// TIA Portal project "2020-11-06_gestioneMotoreJogSS" (V16)
// Programma che gestisce la ventilazione di un motore

(* hardware
DEVICE "Stazione SIMATIC 1200_1"  S71200.Device
   slot 0: "Telaio di montaggio S7-1200"  Rack  V1.0
   slot 1: "PLC_1"  CPU 1215C DC/DC/DC  6ES7 215-1AG40-0XB0  V4.2
*)

// ===== PLC "PLC_1"  CPU 1215C DC/DC/DC =====

VAR_GLOBAL   // PLC tag table "Tabella delle variabili standard"
   "ventA_f" AT %I0.0 : Bool;
   "ventB_f" AT %I0.1 : Bool;
   "ventC_f" AT %I0.2 : Bool;
   "pulsanteJog_f" AT %I0.3 : Bool;
   "pulsanteStart_f" AT %I0.4 : Bool;
   "pulsanteStop_f" AT %I0.5 : Bool;
   "modoJog_f" AT %I0.6 : Bool;
   "motore" AT %Q0.0 : Bool;
   "ventilaz_NOOK" AT %Q0.1 : Bool;
   "modoSS_f" AT %I0.7 : Bool;
   "out2" AT %Q0.2 : Bool;
   "out3" AT %Q0.3 : Bool;
   "out4" AT %Q0.4 : Bool;
   "sempre vero" AT %M6.0 : Bool;   // bit sempre vero
   "uscite byte" AT %QB0 : Byte;   // Uscite fisiche
   "uscite memorie" AT %MB1 : Byte;   // uscite memorie da usare come ingressi
   "out4_M" AT %M1.4 : Bool;
   "out3_M" AT %M1.3 : Bool;
   "out2_M" AT %M1.2 : Bool;
   "ventilaz_NOOK_M" AT %M1.1 : Bool;
   "motore_M" AT %M1.0 : Bool;
   "ingressi byte" AT %IB0 : Byte;   // Ingressi fisici
   "ingressi memorie" AT %MB0 : Byte;   // Ingressi Na non filtrati
   "in0_na" AT %M0.0 : Bool;
   "in1_na" AT %M0.1 : Bool;
   "in2_na" AT %M0.2 : Bool;
   "in3_na" AT %M0.3 : Bool;
   "in4_na" AT %M0.4 : Bool;
   "in5_na" AT %M0.5 : Bool;
   "in6_na" AT %M0.6 : Bool;
   "in7_na" AT %M0.7 : Bool;
   "out5" AT %Q0.5 : Bool;
   "out6" AT %Q0.6 : Bool;
   "out7" AT %Q0.7 : Bool;
   "out5_M" AT %M1.5 : Bool;
   "out6_M" AT %M1.6 : Bool;
   "out7_M" AT %M1.7 : Bool;
   "ingressi memorie filtrato" AT %MB2 : Byte;
   "ventA" AT %M2.0 : Bool;
   "ventB" AT %M2.1 : Bool;
   "ventC" AT %M2.2 : Bool;
   "pulsanteJog" AT %M2.3 : Bool;
   "pulsanteStart" AT %M2.4 : Bool;
   "pulsanteStop" AT %M2.5 : Bool;
   "modoJog" AT %M2.6 : Bool;
   "modoSS" AT %M2.7 : Bool;
   "ingressi memorie_p" AT %MB3 : Byte;
   "in0_p" AT %M3.0 : Bool;
   "in1_p" AT %M3.1 : Bool;
   "in2_p" AT %M3.2 : Bool;
   "in3_p" AT %M3.3 : Bool;
   "pulsanteStart_p" AT %M3.4 : Bool;
   "pulsanteStop_p" AT %M3.5 : Bool;
   "in6_p" AT %M3.6 : Bool;
   "in7_p" AT %M3.7 : Bool;
   "ingressi_memorie_var_p" AT %MB4 : Byte;
   "in0_var_p" AT %M4.0 : Bool;
   "in1_var_p" AT %M4.1 : Bool;
   "in2_var_p" AT %M4.2 : Bool;
   "in3_var_p" AT %M4.3 : Bool;
   "in4_var_p" AT %M4.4 : Bool;
   "in5_var_p" AT %M4.5 : Bool;
   "in6_var_p" AT %M4.6 : Bool;
   "in7_var_p" AT %M4.7 : Bool;
   "ventilazione_OK" AT %M10.0 : Bool;
   "modoJog_OK" AT %M10.1 : Bool;
   "modoSS_OK" AT %M10.2 : Bool;
   "motoreJog" AT %M10.3 : Bool;
   "motoreSS" AT %M10.4 : Bool;
END_VAR

VAR_GLOBAL CONSTANT   // PLC tag table "Tabella delle variabili standard"
   "maschera NCNA" : Byte := B#2#00100100;   // mettere a 1 i bit NC
   "filtro in0" : Time := T#500ms;
   "filtro in1" : Time := T#500ms;
   "filtro in2" : Time := T#500ms;
   "filtro in3" : Time := T#200ms;
   "filtro in4" : Time := T#500ms;
   "filtro in5" : Time := T#100ms;
   "filtro in6" : Time := T#1s;
   "filtro in7" : Time := T#1s;
   "Maschera Out Reset" : Byte := B#2#00000000;
END_VAR

// folder: System blocks/Program resources

DATA_BLOCK "filtro_in0"   // DB1
{ S7_Optimized_Access := 'TRUE' }
AUTHOR : Simatic
FAMILY : IEC
NAME : IEC_TMR
VERSION : 1.0
// stored: InstanceOfName IEC_TIMER
"IEC_TIMER"
BEGIN
END_DATA_BLOCK

DATA_BLOCK "filtro_in1"   // DB2
{ S7_Optimized_Access := 'TRUE' }
AUTHOR : Simatic
FAMILY : IEC
NAME : IEC_TMR
VERSION : 1.0
// stored: InstanceOfName IEC_TIMER
"IEC_TIMER"
BEGIN
END_DATA_BLOCK

DATA_BLOCK "filtro_in2"   // DB3
{ S7_Optimized_Access := 'TRUE' }
AUTHOR : Simatic
FAMILY : IEC
NAME : IEC_TMR
VERSION : 1.0
// stored: InstanceOfName IEC_TIMER
"IEC_TIMER"
BEGIN
END_DATA_BLOCK

DATA_BLOCK "filtro_in3"   // DB4
{ S7_Optimized_Access := 'TRUE' }
AUTHOR : Simatic
FAMILY : IEC
NAME : IEC_TMR
VERSION : 1.0
// stored: InstanceOfName IEC_TIMER
"IEC_TIMER"
BEGIN
END_DATA_BLOCK

DATA_BLOCK "filtro_in4"   // DB5
{ S7_Optimized_Access := 'TRUE' }
AUTHOR : Simatic
FAMILY : IEC
NAME : IEC_TMR
VERSION : 1.0
// stored: InstanceOfName IEC_TIMER
"IEC_TIMER"
BEGIN
END_DATA_BLOCK

DATA_BLOCK "filtro_in5"   // DB6
{ S7_Optimized_Access := 'TRUE' }
AUTHOR : Simatic
FAMILY : IEC
NAME : IEC_TMR
VERSION : 1.0
// stored: InstanceOfName IEC_TIMER
"IEC_TIMER"
BEGIN
END_DATA_BLOCK

DATA_BLOCK "filtro_in6"   // DB7
{ S7_Optimized_Access := 'TRUE' }
AUTHOR : Simatic
FAMILY : IEC
NAME : IEC_TMR
VERSION : 1.0
// stored: InstanceOfName IEC_TIMER
"IEC_TIMER"
BEGIN
END_DATA_BLOCK

DATA_BLOCK "filtro_in7"   // DB8
{ S7_Optimized_Access := 'TRUE' }
AUTHOR : Simatic
FAMILY : IEC
NAME : IEC_TMR
VERSION : 1.0
// stored: InstanceOfName IEC_TIMER
"IEC_TIMER"
BEGIN
END_DATA_BLOCK

// folder: (top level)

FUNCTION "Ingressi e uscite" : Void   // FC1, LAD
{ S7_Optimized_Access := 'TRUE' }
VERSION : 0.1
   VAR_TEMP   // added for the SCL form of the ladder/FBD networks
      _w1 : Bool;
   END_VAR
BEGIN

REGION Network 1: creazione immagine uscite (MB1) da usare come ingressi
   // creazione immagine uscite (MB1) da usare come ingressi
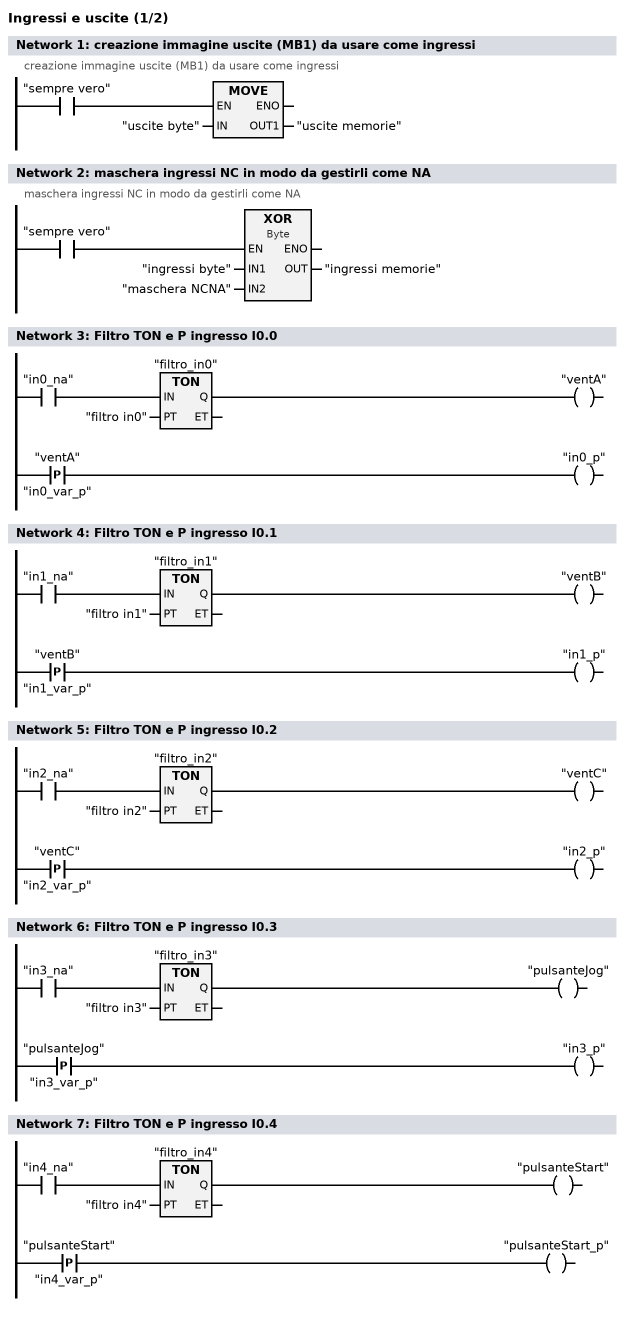
   RUNG wire#powerrail
      Contact( "sempre vero" )
      { S7_GenerateENO := "TRUE" } Move(in := "uscite byte", out1 => "uscite memorie")
   END_RUNG
   // the same network as SCL:
   IF "sempre vero" THEN "uscite memorie" := "uscite byte"; END_IF;
END_REGION

REGION Network 2: maschera ingressi NC in modo da gestirli come NA
   // maschera ingressi NC in modo da gestirli come NA
   IF "sempre vero" THEN "ingressi memorie" := "ingressi byte" XOR "maschera NCNA"; END_IF;
END_REGION

REGION Network 3: Filtro TON e P ingresso I0.0
   "filtro_in0".TON(IN := "in0_na", PT := "filtro in0");
   "ventA" := "filtro_in0".Q;
   #_w1 := "ventA" AND NOT "in0_var_p";   // rising edge of "ventA"
   "in0_var_p" := "ventA";
   "in0_p" := #_w1;
END_REGION

REGION Network 4: Filtro TON e P ingresso I0.1
   "filtro_in1".TON(IN := "in1_na", PT := "filtro in1");
   "ventB" := "filtro_in1".Q;
   #_w1 := "ventB" AND NOT "in1_var_p";   // rising edge of "ventB"
   "in1_var_p" := "ventB";
   "in1_p" := #_w1;
END_REGION

REGION Network 5: Filtro TON e P ingresso I0.2
   "filtro_in2".TON(IN := "in2_na", PT := "filtro in2");
   "ventC" := "filtro_in2".Q;
   #_w1 := "ventC" AND NOT "in2_var_p";   // rising edge of "ventC"
   "in2_var_p" := "ventC";
   "in2_p" := #_w1;
END_REGION

REGION Network 6: Filtro TON e P ingresso I0.3
   "filtro_in3".TON(IN := "in3_na", PT := "filtro in3");
   "pulsanteJog" := "filtro_in3".Q;
   #_w1 := "pulsanteJog" AND NOT "in3_var_p";   // rising edge of "pulsanteJog"
   "in3_var_p" := "pulsanteJog";
   "in3_p" := #_w1;
END_REGION

REGION Network 7: Filtro TON e P ingresso I0.4
   "filtro_in4".TON(IN := "in4_na", PT := "filtro in4");
   "pulsanteStart" := "filtro_in4".Q;
   #_w1 := "pulsanteStart" AND NOT "in4_var_p";   // rising edge of "pulsanteStart"
   "in4_var_p" := "pulsanteStart";
   "pulsanteStart_p" := #_w1;
END_REGION

REGION Network 8: Filtro TON e P ingresso I0.5
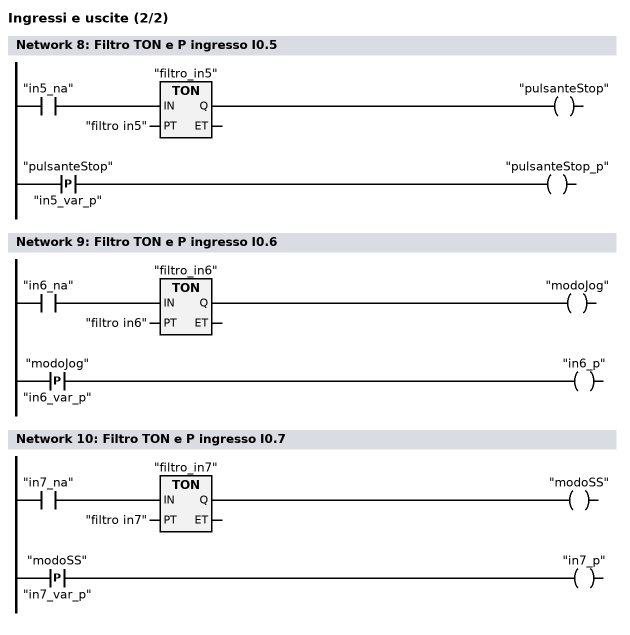
   "filtro_in5".TON(IN := "in5_na", PT := "filtro in5");
   "pulsanteStop" := "filtro_in5".Q;
   #_w1 := "pulsanteStop" AND NOT "in5_var_p";   // rising edge of "pulsanteStop"
   "in5_var_p" := "pulsanteStop";
   "pulsanteStop_p" := #_w1;
END_REGION

REGION Network 9: Filtro TON e P ingresso I0.6
   "filtro_in6".TON(IN := "in6_na", PT := "filtro in6");
   "modoJog" := "filtro_in6".Q;
   #_w1 := "modoJog" AND NOT "in6_var_p";   // rising edge of "modoJog"
   "in6_var_p" := "modoJog";
   "in6_p" := #_w1;
END_REGION

REGION Network 10: Filtro TON e P ingresso I0.7
   "filtro_in7".TON(IN := "in7_na", PT := "filtro in7");
   "modoSS" := "filtro_in7".Q;
   #_w1 := "modoSS" AND NOT "in7_var_p";   // rising edge of "modoSS"
   "in7_var_p" := "modoSS";
   "in7_p" := #_w1;
END_REGION
END_FUNCTION

ORGANIZATION_BLOCK "Main"   // OB1, LAD, ProgramCycle
TITLE = "Main Program Sweep (Cycle)"
{ S7_Optimized_Access := 'TRUE' }
VERSION : 0.1
// Programma da copiare e incollare ed editare per raggiungere le funzionalità desiderate
// Caratteristiche:
// - Predisposizione delle variabili in OB100 (programma che si avvia una sola volta al reset)
// - Generazione di variabili di appoggio degli ingressi in logica vera (maschera NANC) e filtrati secondo la predisposizione di apposite costanti
// - Generazione di variabili di appoggio relative ai fronti di salita degli ingressi in logica vera (maschera NANC) e filtrati secondo la predisposizione di apposite costanti
// - Generazione di variabili di appoggio delle uscite alla fine del ciclo precedente, da poter essere utilizzate per interrogazioni con valore costante per quel ciclo
// - Uso dell'FC non parametrico Ingresso e Uscite
// 
// ISTRUZIONI D'USO
// 
// 1. Sezione COSTANTI. Aggiornare:
// - maschera NCNA (ricordarsi che il bit 0 è quello più a destra e che si inserisce 1 se NC e 0 se NA)
// - valori dei filtri (se no filtro inserire 1ms)
// Dichiarare altre eventuali costanti
// 
// 2. Sezione VARIABILI. Dare nomi appropriati a:
// - OUTx (Q0.x) e OUTx_M (M1.x)
// - Inx (M2.x) e Inx_p (M3.x)
// Dichiarare altre eventuali variabili
// 
// 3. Rimuovere il segmento 2 e aggiungere i nuovi segmenti su MAIN SENZA MODIFICARE IL SEGMENTO 1 e SENZA MODIFICARE IL BLOCCO FC1 Ingressi e Uscite
BEGIN

REGION Network 1: richiamo FC
   // creazione immagine uscite (MB1) da usare come ingressi
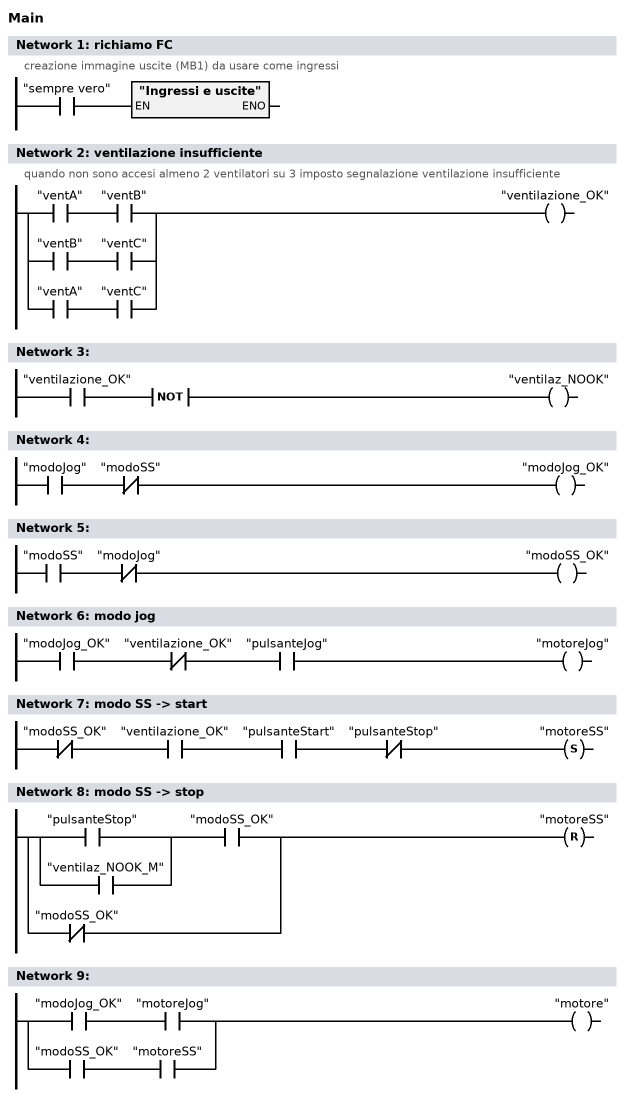
   RUNG wire#powerrail
      Contact( "sempre vero" )
      "Ingressi e uscite"()
   END_RUNG
   // the same network as SCL:
   IF "sempre vero" THEN "Ingressi e uscite"(); END_IF;
END_REGION

REGION Network 2: ventilazione insufficiente
   // quando non sono accesi almeno 2 ventilatori su 3 imposto segnalazione ventilazione insufficiente
   RUNG wire#powerrail
      Contact( "ventA" )
      Contact( "ventB" )
      wire#w1
      Coil( "ventilazione_OK" )
   END_RUNG
   RUNG wire#powerrail
      Contact( "ventB" )
      Contact( "ventC" )
   END_RUNG wire#w1
   RUNG wire#powerrail
      Contact( "ventA" )
      Contact( "ventC" )
   END_RUNG wire#w1
   // the same network as SCL:
   "ventilazione_OK" := ("ventA" AND "ventB") OR ("ventB" AND "ventC") OR ("ventA" AND "ventC");
END_REGION

REGION Network 3
   RUNG wire#powerrail
      Contact( "ventilazione_OK" )
      Not()
      Coil( "ventilaz_NOOK" )
   END_RUNG
   // the same network as SCL:
   "ventilaz_NOOK" := NOT "ventilazione_OK";
END_REGION

REGION Network 4
   RUNG wire#powerrail
      Contact( "modoJog" )
      I_Contact( "modoSS" )
      Coil( "modoJog_OK" )
   END_RUNG
   // the same network as SCL:
   "modoJog_OK" := "modoJog" AND NOT "modoSS";
END_REGION

REGION Network 5
   RUNG wire#powerrail
      Contact( "modoSS" )
      I_Contact( "modoJog" )
      Coil( "modoSS_OK" )
   END_RUNG
   // the same network as SCL:
   "modoSS_OK" := "modoSS" AND NOT "modoJog";
END_REGION

REGION Network 6: modo jog
   RUNG wire#powerrail
      Contact( "modoJog_OK" )
      I_Contact( "ventilazione_OK" )
      Contact( "pulsanteJog" )
      Coil( "motoreJog" )
   END_RUNG
   // the same network as SCL:
   "motoreJog" := "modoJog_OK" AND NOT "ventilazione_OK" AND "pulsanteJog";
END_REGION

REGION Network 7: modo SS -> start
   RUNG wire#powerrail
      I_Contact( "modoSS_OK" )
      Contact( "ventilazione_OK" )
      Contact( "pulsanteStart" )
      I_Contact( "pulsanteStop" )
      S_Coil( "motoreSS" )
   END_RUNG
   // the same network as SCL:
   IF NOT "modoSS_OK" AND "ventilazione_OK" AND "pulsanteStart" AND NOT "pulsanteStop" THEN
       "motoreSS" := TRUE;
   END_IF;
END_REGION

REGION Network 8: modo SS -> stop
   RUNG wire#powerrail
      Contact( "pulsanteStop" )
      wire#w1
      Contact( "modoSS_OK" )
      wire#w2
      R_Coil( "motoreSS" )
   END_RUNG
   RUNG wire#powerrail
      Contact( "ventilaz_NOOK_M" )
   END_RUNG wire#w1
   RUNG wire#powerrail
      I_Contact( "modoSS_OK" )
   END_RUNG wire#w2
   // the same network as SCL:
   IF (("pulsanteStop" OR "ventilaz_NOOK_M") AND "modoSS_OK") OR NOT "modoSS_OK" THEN
       "motoreSS" := FALSE;
   END_IF;
END_REGION

REGION Network 9
   RUNG wire#powerrail
      Contact( "modoJog_OK" )
      Contact( "motoreJog" )
      wire#w1
      Coil( "motore" )
   END_RUNG
   RUNG wire#powerrail
      Contact( "modoSS_OK" )
      Contact( "motoreSS" )
   END_RUNG wire#w1
   // the same network as SCL:
   "motore" := ("modoJog_OK" AND "motoreJog") OR ("modoSS_OK" AND "motoreSS");
END_REGION
END_ORGANIZATION_BLOCK

ORGANIZATION_BLOCK "Startup"   // OB100, LAD, Startup
TITLE = "Complete Restart"
{ S7_Optimized_Access := 'TRUE' }
VERSION : 0.1
   VAR_INPUT
      LostRetentive : Bool;   // True if retentive data are lost
      LostRTC : Bool;   // True if real time clock is lost
   END_VAR
BEGIN

REGION Network 1: bit sempre vero
   // creazione bit sempre vero
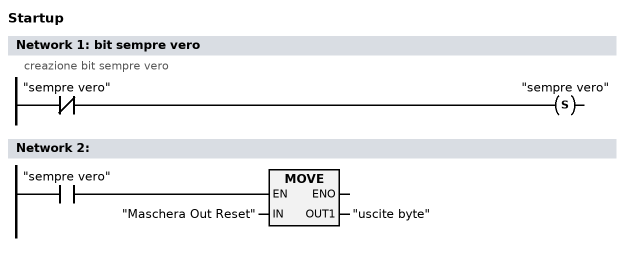
   RUNG wire#powerrail
      I_Contact( "sempre vero" )
      S_Coil( "sempre vero" )
   END_RUNG
   // the same network as SCL:
   IF NOT "sempre vero" THEN "sempre vero" := TRUE; END_IF;
END_REGION

REGION Network 2
   RUNG wire#powerrail
      Contact( "sempre vero" )
      { S7_GenerateENO := "TRUE" } Move(in := "Maschera Out Reset", out1 => "uscite byte")
   END_RUNG
   // the same network as SCL:
   IF "sempre vero" THEN "uscite byte" := "Maschera Out Reset"; END_IF;
END_REGION
END_ORGANIZATION_BLOCK